FUNCTION_BLOCK FB_MER EXTENDS FB_CtrlBase IMPLEMENTS IBuffer
VAR_INPUT
	/// Sensor hanger detected
	In_bolHangerDetected: BOOL;
	/// Pin of Drive is detected
	In_bolPinDetected: BOOL;
	/// Sensors for jam detection
	In_a_bolJamSensor: ARRAY[1..cMAX_JAM_SENSORS] OF BOOL;
END_VAR
VAR
	/// Specific interface struct for public access
	SIf: T_Ctrl_SIf_MER;
	/// List of pointers to Childs
	a_pLineChildCtrl: ARRAY[0..Base_Const.cMaxNrOfChilds] OF POINTER TO FB_SLB;
	/// List of childs common interface
	a_pLineChildCIF: ARRAY[0..Base_Const.cMaxNrOfChilds] OF POINTER TO T_Ctrl_CIf;
	/// List of childs specific interface for additional parameters or cur
	a_pLineChildSIF: ARRAY[0..Base_Const.cMaxNrOfChilds] OF POINTER TO T_Ctrl_SIf_SLB;
	/// Function specific variables
	usiNumOfLines: USINT;
	usiNumOfValidPointerToLine: USINT;
	bolHangerExist: BOOL;
	bolGoToRun: BOOL;
	dinPassedTotalLineXOld: DINT;
	/// Used for counting passed hangers if "E_Typ_MER_MODE.MergeOverSetpoint" is selected.
	dinNumOfPassedHangers: DINT;
	/// Used for time measurement if "E_Typ_MER_MODE.MergeOverTime" is selected.
	udiMergingTime: UDINT;
	usiLineNumToReleaseAll: USINT;
	usiIndexToRelease: USINT;
	/// Last new position value from parent
	dinTransportPositionOld_um: DINT;
	/// Driven Way in the task
	dinDrivenWay_um: DINT;
	/// Position correction in faster Task cycletime
	dinPositionCorrection_um: DINT;
	/// Position of the section
	dinPositionSection_um: DINT;
	/// Section buffer
	a_stSectionBuffer: ARRAY[0..cusiSectionBuffer_SIZE] OF T_MER_Buffer_Sections;
	/// Edge detection of the inputs
	bolRE_HangerDetected: BOOL;
	/// Pin of Drive is detected
	bolRE_PinDetected: BOOL;
	bolModeMergeIntoTrpUsed: BOOL;
	bolSectionFree: BOOL;
	bolReleaseHanger: BOOL;
	/// Used to detect if a section is driven out
	dinPositionOfLastLine_um: DINT;
	/// Shadow copy of In_a_bolJamSensor[]
	a_bolJamSensorOnce: ARRAY[1..cMAX_JAM_SENSORS] OF BOOL;
	/// Start time of jam sensor is true
	a_udiTimeJamDetection: ARRAY[1..cMAX_JAM_SENSORS] OF UDINT;
	/// Jam at merger output detected 
	bolJamDetected: BOOL;
	/// Loop variable
	intI: INT;
	/// Simulated section length
	dinSimSectionLength_um: DINT := 510000;
	/// Simulated way to trigger section start/end
	dinSimWayTrigSection_um: DINT;
END_VAR
VAR CONSTANT
	/// sub States
	cSTA_SUB_INITIALIZED: INT := 500;
	cSTA_SUB_WAIT_FOR_CMD: INT := 502;
	cSTA_SUB_CHECK_HANGER_EXIST: INT := 504;
	cSTA_SUB_SEND_RELEASE: INT := 506;
	cSTA_SUB_SEND_RELEASE_ALL: INT := 508;
	cSTA_SUB_SEND_STOP: INT := 510;
	cSTA_SUB_WAIT_JOB_DONE: INT := 512;
	cSTA_SUB_CHECK_MERGE_CON: INT := 514;
	cSTA_SUB_WAIT_LINE_FREE: INT := 516;
	cSTA_SUB_END: INT := 518;
END_VAR

(*__________________________________________________________________________________________________
¦	
¦	Vistaprint Schweiz GmbH
¦	CH - 8401 Winterthur
¦
¦	www.vistaprint.ch - info@vistaprint.ch
¦___________________________________________________________________________________________________

Function desription:
The controller automatically merge hangers from different lines dependent time or distribution of the number of hangers.
Lines are always from controller type slide buffer FB_SLB.

History:
Version		Date			Author		Comment
---------------------------------------------------------------------------------------------------
0.00.1		05.09.2013		AVME/DSC	Start history. 
0.00.2		09.09.2013		AVME/DSC 	Integration of all merger basic functionalities. Test on simulator.
										Controller can work in 2 different main modes:
										-> "automatic", controller automatically merge hangers from different lines dependent E_Typ_MER_AUTO_MODE
										-> "on command", in case if merger work as charge controller. Release line X dependent from parent command.
0.00.3		19.09.2013		AVME/PRE	Implement new Base Concept
0.00.4		01.10.2013		AVME/DSC	Sub state machine general handling deleted. Not used anymore. Handled in Base Class.										
0.00.5		03.10.2013		AVME/PRE	Integrate new function insert Belt		
0.00.6		03.10.2013		AVME/PRE	Insert new sub state LOCK_SECTION.	
0.00.7		15.10.2013		AVME/DSC	Complete redesign of the merger "MergeIntoTrp" mode.
0.00.8		30.10.2013		AVME/DSC	Modifications for "MergeIntoTrp" mode during test at the tool. Good merging possible with drive speed = 0. (slow speed)
										Merging with higher speed not possible!				
0.00.9		08.11.2013		AVME/MRU	Stop merger if outfeed sensor detect a jam (Bugzilla Nr. 8)
0.00.10		03.12.2013		AVME/MRU	Add MaxCapacity / NumOfHangers properties
0.00.11		09.12.2013		AVME/DSC	Modification in method "checkStateAllLines".
										Special condition: In case if the child is in state ERROR and STOP is requested. Set child as checked.
										Parent controller need state STOP that automatic stop sequence can work for all other childs.
0.00.12		13.01.2014		AVME/MRU	Bugzilla ID 03: BufferFull for LineControl added

__________________________________________________________________________________________________*)


IF ((me.bolActivate) AND (THIS^.checkChildValid())) THEN // cyclic call enabled
	IF (CIf.Info.bolInitDone=FALSE) THEN // first cycle -> init
		CtrlInit();
		CIf.Info.bolInitDone := TRUE;
	ELSE
		CycleStartDuty();
	
		Always();
		
		StateMachine();
		
		CycleEndDuty();
	END_IF
END_IF;

METHOD PROTECTED sta_OFF : BOOL
// state implemetation
//--------------------------------------------------------------------------------------
// Entry action
	IF (me.StateMachine.intState<>me.StateMachine.intStateLastCycle) THEN
		me.StateMachine.intStateLastCycle := me.StateMachine.intState;
		;		
	END_IF

//--------------------------------------------------------------------------------------
// Cyclic action
	IF (me.StateMachine.intState=me.StateMachine.intStateLastCycle) THEN
		
		// Reset total counter
		SIf.Cur.dinNumOfMergedHangersTotal:= 0;
		
		// State Change Condition
		IF (me.Alarm.eActivAlmClass<>E_AlmClass.EOFF) AND (me.Alarm.eActivAlmClass<>E_AlmClass.OFF) THEN
			IF (me.intCmd=cCMD_STOP) THEN
				me.StateMachine.intStateNext := cSTA_STOPBusy;
			ELSIF (me.intCmd=cCMD_RUN) THEN 
				me.StateMachine.intStateNext := cSTA_RUNBusy;
			END_IF
		END_IF
	END_IF

//--------------------------------------------------------------------------------------
// Exit action
	IF (me.StateMachine.intState<>me.StateMachine.intStateNext) THEN
		;
	END_IF
END_METHOD

METHOD PROTECTED StateMachine : BOOL
SUPER^.StateMachine();

// main statemachine of base controller
CASE me.StateMachine.intState OF
    cSTA_STOPBusy: 
        THIS^.sta_STOPBusy();
    cSTA_STOP: 
        THIS^.sta_STOP();
	cSTA_RUNBusy: 
        THIS^.sta_RUNBusy();
    cSTA_RUN: 
        THIS^.sta_RUN();				
END_CASE;
END_METHOD

METHOD PROTECTED checkStateAllLines : BOOL
VAR_INPUT
	cSTA: INT;
END_VAR
VAR
	ii: INT;
	usiNumOfCheckedChilds: USINT;
END_VAR
// Method check input state of all lines

//Init
checkStateAllLines:= FALSE;
usiNumOfCheckedChilds:= 0;

// Loop over all childs
FOR ii:=0 TO usiNumOfLines-1 BY 1 DO
	// Check state	
	// Special condition: In case if the child is in state ERROR and STOP is requested. Set child as checked.
	// Parent controller need state STOP that automatic stop sequence can work for all other childs.
	IF (a_pLineChildCIF[ii]^.Job.intState = cSTA) OR ((a_pLineChildCIF[ii]^.Job.intState = cSTA_ERROR) AND (cSTA = cSTA_STOP)) THEN
		usiNumOfCheckedChilds:= usiNumOfCheckedChilds+1;
		SIf.Cur.a_bolChildReady[ii] := TRUE;
	ELSE
		SIf.Cur.a_bolChildReady[ii] := FALSE;		
	END_IF

END_FOR

// All states equal the input state
IF (usiNumOfCheckedChilds = usiNumOfLines) THEN
	checkStateAllLines:= TRUE;
END_IF
END_METHOD

METHOD PROTECTED getCmdState : STRING
VAR_INPUT
	intCmdState: INT;
	bolState: BOOL;
END_VAR
getCmdState := SUPER^.getCmdState(intCmdState:=intCmdState,bolState:=bolState); // get global/base defined cmds/states
IF (getCmdState='') THEN // global not defined get local
	// get string cmd/state string information in runtime
	IF (bolState=FALSE) THEN
		// cmd's
		CASE intCmdState OF
		END_CASE;
	ELSE
	
	// states
		CASE intCmdState OF	
			// SUB States
			cSTA_SUB_INITIALIZED:
				getCmdState := 'cSTA_SUB_INITIALIZED';			
			cSTA_SUB_WAIT_FOR_CMD:
				getCmdState := 'cSTA_SUB_WAIT_FOR_CMD';					
			cSTA_SUB_CHECK_HANGER_EXIST:
				getCmdState := 'cSTA_SUB_CHECK_HANGER_EXIST';
			cSTA_SUB_SEND_RELEASE:
				getCmdState := 'cSTA_SUB_SEND_RELEASE';
			cSTA_SUB_SEND_RELEASE_ALL:
				getCmdState := 'cSTA_SUB_SEND_RELEASE_ALL';	
			cSTA_SUB_SEND_STOP:
				getCmdState := 'cSTA_SUB_SEND_STOP';		
			cSTA_SUB_WAIT_JOB_DONE:
				getCmdState := 'cSTA_SUB_WAIT_JOB_DONE';
			cSTA_SUB_CHECK_MERGE_CON:
				getCmdState := 'cSTA_SUB_CHECK_MERGE_CON';
			cSTA_SUB_WAIT_LINE_FREE:
				getCmdState := 'cSTA_SUB_WAIT_LINE_FREE';	
			cSTA_SUB_END:
				getCmdState := 'cSTA_SUB_END';	
		END_CASE;
	END_IF
END_IF
END_METHOD

METHOD FB_init : BOOL
VAR_INPUT
	///if TRUE, the retain variables are initialized (warm start / cold start)
	bInitRetains: BOOL;
	///if TRUE, the instance afterwards gets moved into the copy code (online change)
	bInCopyCode: BOOL;
END_VAR
VAR
	ii: UINT;
END_VAR
//------------------------------------------------------------------------------------------------------------------------
// to manually change in new FUB implementation!!!
// define valid commands for this controller
FOR ii:= 0 TO (SIZEOF(CIf.Job.aCmdList)/SIZEOF(CIf.Job.aCmdList[0])-1) BY 1 DO
	IF (CIf.Job.aCmdList[ii].intCmd=cCMD_INITIALIZED) THEN
		// found first empty array element
		EXIT;
	END_IF
END_FOR

CIf.Job.aCmdList[ii].intCmd := cCMD_STOP;
CIf.Job.aCmdList[ii].strName := 'Stop'; 
CIf.Job.aCmdList[ii].bolAvailable := TRUE;
ii := ii +1;
CIf.Job.aCmdList[ii].intCmd := cCMD_RUN;
CIf.Job.aCmdList[ii].strName := 'Run';
CIf.Job.aCmdList[ii].bolAvailable := TRUE;

// set name of class/typ
CIf.Info.strType := 'FB_MER'; 

// set alarm class
SIf.Alm[1].eAlmClass := E_AlmClass.STOP;
SIf.Alm[1].strText := 'Invalid child pointer';
SIf.Alm[2].eAlmClass := E_AlmClass.INFO;
SIf.Alm[2].strText := 'Invalid line number. Line not exist';
SIf.Alm[3].eAlmClass := E_AlmClass.INFO;
SIf.Alm[3].strText := 'Merger waits for jam sensor free'; 


//*******************************************************************************
// initial values
//*******************************************************************************

// software configuration
CIf.SwCfg.bolExist := TRUE;
CIf.SwCfg.bolSimulation := FALSE;

// configuration
SIf.Cfg.usiMergeMainMode:= E_Typ_MER_MODE.Automatic;
SIf.Cfg.usiCountJamSensors:= 0;

// parameter
SIf.Par.udi_jamTimeout_ms:= 500;
// Default parameter for the lines are set in method InitLines
END_METHOD

METHOD PROTECTED Always : BOOL
VAR
	/// Looping variable
	intSec: INT;
END_VAR
IF (me.bolChangeBackToAUTO=TRUE) THEN // switch mode to automatic switch off controller
	//me.StateMachine.intStateNext := cSTA_OFFBusy;
	//me.bolChangeBackToAUTO := FALSE; // for cylinder no change to off when switch to automatic!!
END_IF

SUPER^.Always();

// ----------------------------------------------------------------------------------
// cyclic actions outside of statemachine
IF (me.StateMachine.intState<>cSTA_SINGLE_ANSWER) THEN
	
	//-------------------------------------------------
	// Provide current values for the parent
	//-------------------------------------------------	
	
	// Number of lines to merge, depends on how many times the method "AddLine" was called at init
	SIf.Cur.usiNumOfLinesToMerge:= usiNumOfLines;
	// Actual Item Count of this controller -> based on all lines
	SIf.Cur.dinCurrentItemCount:= THIS^.CalcSumOfItems();
	// Max. buffer capacity -> based on all lines
	SIf.Cur.dinMaxCapacity:= THIS^.CalcMaxCapacity();	
	
	
	// Check if mode "MergeIntoTrp" is configured. 
	// If one line is configured with this mode, all other lines will be set to the same mode automatically in CtrlInit. Mixed mode not possible.
	IF ((SIf.Cfg.usiMergeMainMode = E_Typ_MER_MODE.Automatic) AND (SIf.Par.a_LinePar[0].usiMergeMode = E_Typ_MER_AUTO_MODE.MergeIntoTrp)) THEN
	
		//----------------------------------------------------------------------
		// Calculate position for transport 
		//----------------------------------------------------------------------
			
		// If this task is used in a faster cycle as the parent, the driven way will be indirectly calculated (synchronized) over the transport speed.
		// If transport position changed from the parent (new value), synchronize the driven way 
		
		IF (dinTransportPositionOld_um <> SIf.Cur.dinTransportPosition_um) THEN
			dinDrivenWay_um := SIf.Cur.dinTransportPosition_um - SIf.Cur.dinTransportPositionCalc_um;
			SIf.Cur.dinTransportPositionCalc_um := SIf.Cur.dinTransportPosition_um;
			dinTransportPositionOld_um := SIf.Cur.dinTransportPosition_um;
			dinPositionCorrection_um := 0;
		ELSE
			// During the time, if there is no position change from the parent, calculate the driven way dependent the speed of transport.		
			// s = v * t
			dinDrivenWay_um := LREAL_TO_DINT(DINT_TO_LREAL(SIf.Cur.dinTransportspeed_um_s) * UDINT_TO_LREAL(me.FUBInfo.udiSample_ms) / 1000.0 );
			dinPositionCorrection_um := dinPositionCorrection_um + dinDrivenWay_um;
			SIf.Cur.dinTransportPositionCalc_um := dinTransportPositionOld_um + dinPositionCorrection_um;
		END_IF
	
	END_IF
	
END_IF

// ----------------------------------------------------------------------------------
// Always change actions in Base Library
// ----------------------------------------------------------------------------------
// overrule error always from base -> no EOFF State!! in EOFF go to OFF
IF (me.StateMachine.intStateNext = cSTA_EOFFBusy) THEN
	IF (me.StateMachine.intState=cSTA_OFF) THEN
		me.StateMachine.intStateNext := cSTA_OFF;
	ELSE // stay in OFF
		me.StateMachine.intStateNext := cSTA_OFFBusy;
	END_IF
END_IF

// Conditions Always
IF (((me.Alarm.eActivAlmClass=E_AlmClass.EOFF) OR (me.Alarm.eActivAlmClass=E_AlmClass.OFF) OR (me.intCmd=cCMD_OFF))
		 AND (me.StateMachine.intState<>cSTA_ERROR) AND (me.StateMachine.intState<>cSTA_ERRORQuit) AND
		(me.StateMachine.intState<>cSTA_OFF) AND (me.StateMachine.intState<>cSTA_OFFBusy)) THEN
	// alarm evt EOFF, OFF or cmd off
	me.StateMachine.intStateNext := cSTA_OFFBusy;
END_IF
END_METHOD

METHOD PROTECTED IoInBridge : BOOL
// digitale and analoge inputs read from hardware or forcing
SIf.In.bolHangerDetected.map := THIS^.In_bolHangerDetected;
SIf.In.bolPinDetected.map := THIS^.In_bolPinDetected;

// Read sensors for waiting if a jam is detected
FOR intI := 1 TO SIf.Cfg.usiCountJamSensors DO
	SIf.In.a_bolJamSensor[intI].map := THIS^.In_a_bolJamSensor[intI];
	IF (CIf.SwCfg.bolSimulation = FALSE) THEN
		getInBol(CIf.Job.bolIoForce,ADR(SIf.In.a_bolJamSensor[intI]));
	END_IF
END_FOR

IF (CIf.SwCfg.bolSimulation = FALSE) THEN
	getInBol(CIf.Job.bolIoForce,ADR(SIf.In.bolHangerDetected));
	getInBol(CIf.Job.bolIoForce,ADR(SIf.In.bolPinDetected));
	//ctrl.In.bol_PosSwitchBasicDefTyp.intern := getInBol(ctrl.ifc.Job.bol_Force ,ADR(ctrl.In.bol_PosSwitchBasicDefTyp);
ELSE
	//simulation of global IO
END_IF
END_METHOD

METHOD PROTECTED sta_STOPBusy : BOOL
// state implemetation
//--------------------------------------------------------------------------------------
// Entry action
	IF (me.StateMachine.intState<>me.StateMachine.intStateLastCycle) THEN
		me.StateMachine.intStateLastCycle := me.StateMachine.intState;
		
		// send command STOP to all existing line child controller.
		THIS^.CmdToAllLines(cCMD_STOP);

	END_IF

//--------------------------------------------------------------------------------------
// Cyclic action
	IF (me.StateMachine.intState=me.StateMachine.intStateLastCycle) THEN
			
		// State Change Condition
		// Check if all STOPPED
		IF (THIS^.checkStateAllLines(cSTA_STOP)) THEN
			me.StateMachine.intStateNext := cSTA_STOP;
		END_IF
	END_IF

//--------------------------------------------------------------------------------------
// Exit action
	IF (me.StateMachine.intState<>me.StateMachine.intStateNext) THEN
		;
	END_IF
END_METHOD

METHOD PROTECTED CtrlInit : BOOL
VAR
	ii: INT;
END_VAR
SUPER^.CtrlInit();

//----------------------------------------------------------------------
// Initialize all lines
//----------------------------------------------------------------------

// Method initialize all line child controller.
FOR ii:=0 TO usiNumOfLines-1 BY 1 DO	
	a_pLineChildCIF[ii] := THIS^.AddChild(a_pLineChildCtrl[ii]^);
	a_pLineChildSIF[ii] := a_pLineChildCtrl[ii]^.getCtrlSIf();
END_FOR

//----------------------------------------------------------------------
// Check about invalid configuration
//----------------------------------------------------------------------

// Check about invalid configuration of "MergeIntoTrp" mode. If one line is configured with this mode, set all other lines to the same mode.
bolModeMergeIntoTrpUsed:= FALSE;
// Check if any line is configured with "MergeIntoTrp" mode.
FOR ii:= 0 TO (usiNumOfLines-1) DO
	IF (SIf.Par.a_LinePar[ii].usiMergeMode = E_Typ_MER_AUTO_MODE.MergeIntoTrp) THEN
		// Mode is used
		bolModeMergeIntoTrpUsed:= TRUE;
		EXIT;
	END_IF
END_FOR
// Set  all other lines to "MergeIntoTrp" mode.
IF (bolModeMergeIntoTrpUsed = TRUE) THEN
	FOR ii:= 0 TO (usiNumOfLines-1) DO
		SIf.Par.a_LinePar[ii].usiMergeMode:= E_Typ_MER_AUTO_MODE.MergeIntoTrp;
	END_FOR	
END_IF

//----------------------------------------------------------------------
// Determine position of the last line
//----------------------------------------------------------------------
dinPositionOfLastLine_um:= SIf.Par.a_LinePar[usiNumOfLines-1].dinLinePosition_um;
END_METHOD

METHOD PROTECTED sta_STOP : BOOL
// state implemetation
//--------------------------------------------------------------------------------------
// Entry action
	IF (me.StateMachine.intState<>me.StateMachine.intStateLastCycle) THEN
		me.StateMachine.intStateLastCycle := me.StateMachine.intState;
		;
	END_IF

//--------------------------------------------------------------------------------------
// Cyclic action
	IF (me.StateMachine.intState=me.StateMachine.intStateLastCycle) THEN

		// State Change Condition	
		IF (me.intCmd = cCMD_RUN) THEN 
			me.StateMachine.intStateNext := cSTA_RUNBusy;
		END_IF
	END_IF

//-------------------------------------------------------------------------------------
// Exit action
	IF (me.StateMachine.intState<>me.StateMachine.intStateNext) THEN
		;
	END_IF
END_METHOD

METHOD PROTECTED IoOutBridge : BOOL
// digitale and analoge inputs read from hardware or forcing

// ... no physical outputs

IF (CIf.SwCfg.bolSimulation = FALSE) THEN
	// check interlocks to prevent damages
	IF (CIf.Job.bolIlkOverwrite=FALSE) THEN
		;
	END_IF
END_IF
END_METHOD

METHOD PROTECTED CmdToAllLines
VAR_INPUT
	cCMD: INT;
END_VAR
VAR
	ii: INT;
END_VAR
// Method send input command to all existing line child controller.
FOR ii:=0 TO usiNumOfLines-1 BY 1 DO	
	a_pLineChildCIF[ii]^.Job.intACmd:= cCMD;
END_FOR
END_METHOD

METHOD PROTECTED sta_RUN : BOOL
VAR
	/// Looping variable
	intSec: INT;
END_VAR
// state implemetation
//--------------------------------------------------------------------------------------
// Entry action
	IF (me.StateMachine.intState<>me.StateMachine.intStateLastCycle) THEN
		me.StateMachine.intStateLastCycle := me.StateMachine.intState;	
		;	
	END_IF

//--------------------------------------------------------------------------------------
// Cyclic action
	IF (me.StateMachine.intState=me.StateMachine.intStateLastCycle) THEN
			
		//-------------------------------------------------
		// Handling to merge into a transport belt
		//-------------------------------------------------	
		
		// Check if mode "MergeIntoTrp" is configured. 
		// If one line is configured with this mode, all other lines will be set to the same mode automatically in CtrlInit. Mixed mode not possible.
		IF ((SIf.Cfg.usiMergeMainMode = E_Typ_MER_MODE.Automatic) AND (SIf.Par.a_LinePar[0].usiMergeMode = E_Typ_MER_AUTO_MODE.MergeIntoTrp)) THEN
						
			//----------------------------------------------------------------------
			// Set the section start and end positions (triggered by pin sensor)
			//----------------------------------------------------------------------
			
			// Simulation of section start and end
			IF (CIf.SwCfg.bolSimulation = TRUE) THEN		
				SIf.In.bolPinDetected.intern:= FALSE;
				
				IF (dinSimWayTrigSection_um >= dinSimSectionLength_um) THEN
					dinSimWayTrigSection_um:= 0;
					// Set true for one cycle
					SIf.In.bolPinDetected.intern:= TRUE;
				END_IF
				// Increase position		
				dinSimWayTrigSection_um:= dinSimWayTrigSection_um + dinDrivenWay_um;
			END_IF
					
			// Wait for positive edge of the pin sensor (pin detected)
			IF (SIf.In.bolPinDetected.intern = TRUE) AND (bolRE_PinDetected = FALSE) THEN
				bolRE_PinDetected := TRUE;
					
				// Loop over section buffer
				FOR intSec := 0 TO cusiSectionBuffer_SIZE DO
					
					// If start position already set
					IF (a_stSectionBuffer[intSec].usiState = 1) THEN						
						// Set end position of the section
						a_stSectionBuffer[intSec].dinSecEndPos:= 0 - SIf.Par.dinPinLenght_um;
						a_stSectionBuffer[intSec].usiState:= 2;
					END_IF
					
					// Free buffer element  
					IF (a_stSectionBuffer[intSec].usiState = 0) THEN			
						// Set start position of the section
						a_stSectionBuffer[intSec].dinSecStartPos:= 0 - SIf.Par.dinPinLenght_um;
						a_stSectionBuffer[intSec].usiState:= 1;
						EXIT;									  
					END_IF
													
				END_FOR
					
			ELSIF (SIf.In.bolPinDetected.intern = FALSE) AND (bolRE_PinDetected = TRUE) THEN
				bolRE_PinDetected := FALSE;
			END_IF
			
			//----------------------------------------------------------------------
			// Set section engaged (hanger in section)
			//----------------------------------------------------------------------
			
			// Wait for positive edge of the hanger sensor
			IF (SIf.In.bolHangerDetected.intern = TRUE) AND (bolRE_HangerDetected = FALSE) THEN
				bolRE_HangerDetected := TRUE;
					
				// Loop over section buffer to mark buffer element with 3 = section engaged (hanger in section detected by hanger sensor)
				FOR intSec := 0 TO cusiSectionBuffer_SIZE-1 DO		
					
					// Prio 1: Normal sequence.
					IF (SIf.Par.dinHangerSensorPosition_um < a_stSectionBuffer[intSec].dinSecStartPos) AND  
						(SIf.Par.dinHangerSensorPosition_um > (a_stSectionBuffer[intSec].dinSecEndPos - SIf.Par.dinPinLenght_um)) THEN	
							// Mark the buffer element with 3 = section engaged (hanger in section detected by hanger sensor)
							a_stSectionBuffer[intSec].usiState:= 3;
						EXIT;
					
					// Prio 2: If range is not accurately recognized mark buffer element X and X +1.
					ELSIF (SIf.Par.dinHangerSensorPosition_um < a_stSectionBuffer[intSec].dinSecEndPos) AND  
						(SIf.Par.dinHangerSensorPosition_um > a_stSectionBuffer[intSec+1].dinSecStartPos) THEN	
							// Mark the buffer element with 3 = section engaged (hanger in section detected by hanger sensor)
							a_stSectionBuffer[intSec].usiState:= 3;
							a_stSectionBuffer[intSec+1].usiState:= 3;
						EXIT;
					END_IF		
						
				END_FOR	
					
			ELSIF (SIf.In.bolHangerDetected.intern = FALSE) AND (bolRE_HangerDetected = TRUE) THEN
				bolRE_HangerDetected := FALSE;
			END_IF	
				
			//----------------------------------------------------------------------
			// Buffer tracking 
			//----------------------------------------------------------------------
			
			// Move all buffer elements 1 down if hanger was released. State will be set to "0" in state RUN if a hanger is released.
			// Also check if a section is driven out!			
			IF (a_stSectionBuffer[0].usiState = 0) OR (a_stSectionBuffer[0].dinSecEndPos > (dinPositionOfLastLine_um + SIf.Par.dinSectionLenght_um))THEN
				// Loop every buffer element 1 Down
				FOR intSec := 0 TO cusiSectionBuffer_SIZE-1 DO			
					a_stSectionBuffer[intSec].dinSecStartPos := a_stSectionBuffer[intSec+1].dinSecStartPos;
					a_stSectionBuffer[intSec].dinSecEndPos := a_stSectionBuffer[intSec+1].dinSecEndPos;
					a_stSectionBuffer[intSec].dinTrigStartPos := a_stSectionBuffer[intSec+1].dinTrigStartPos;
					a_stSectionBuffer[intSec].dinTrigEndPos := a_stSectionBuffer[intSec+1].dinTrigEndPos;
					a_stSectionBuffer[intSec].usiState := a_stSectionBuffer[intSec+1].usiState;
				END_FOR		
				a_stSectionBuffer[intSec].dinSecStartPos := 0;
				a_stSectionBuffer[intSec].dinSecEndPos := 0;
				a_stSectionBuffer[intSec].dinTrigStartPos := 0;
				a_stSectionBuffer[intSec].dinTrigEndPos := 0;
				a_stSectionBuffer[intSec].usiState := 0;
			END_IF
			
			//----------------------------------------------------------------------
			// Increase positions
			//----------------------------------------------------------------------
				
			// Increase the buffer positions
			FOR intSec := 0 TO cusiSectionBuffer_SIZE DO
				
				IF (a_stSectionBuffer[intSec].usiState = 1) THEN
					// Section start/end
					a_stSectionBuffer[intSec].dinSecStartPos:= a_stSectionBuffer[intSec].dinSecStartPos + dinDrivenWay_um;
					// Trigger start/end
					a_stSectionBuffer[intSec].dinTrigStartPos:= a_stSectionBuffer[intSec].dinSecStartPos - SIf.Par.dinTrigStartOffset_um;
					a_stSectionBuffer[intSec].dinTrigEndPos:= a_stSectionBuffer[intSec].dinSecStartPos - SIf.Par.dinTrigEndOffset_um;	
					
				ELSIF (a_stSectionBuffer[intSec].usiState >= 2) THEN
					// Section start/end
					a_stSectionBuffer[intSec].dinSecStartPos:= a_stSectionBuffer[intSec].dinSecStartPos + dinDrivenWay_um;
					a_stSectionBuffer[intSec].dinSecEndPos:= a_stSectionBuffer[intSec].dinSecEndPos + dinDrivenWay_um;
					// Trigger start/end
					a_stSectionBuffer[intSec].dinTrigStartPos:= a_stSectionBuffer[intSec].dinSecStartPos - SIf.Par.dinTrigStartOffset_um;
					a_stSectionBuffer[intSec].dinTrigEndPos:= a_stSectionBuffer[intSec].dinSecStartPos - SIf.Par.dinTrigEndOffset_um;				
				END_IF
				
			END_FOR	
			
		END_IF
	
		
		// Check States for parent information
		THIS^.checkStateAllLines(cSTA_RUN);

		// Check jam detection
		bolJamDetected := FALSE;
		FOR intI := 1 TO SIf.Cfg.usiCountJamSensors DO
			// Start jam timer
			IF ((SIf.In.a_bolJamSensor[intI].intern = TRUE) AND (a_bolJamSensorOnce[intI] = FALSE)) THEN
				a_bolJamSensorOnce[intI]:= TRUE;
				a_udiTimeJamDetection[intI]:= me.StateMachine.udiTimeInState_ms;
			// Stop jam timer
			ELSIF ((SIf.In.a_bolJamSensor[intI].intern = FALSE) AND (a_bolJamSensorOnce[intI] = TRUE)) THEN
				a_bolJamSensorOnce[intI]:= FALSE;
				//a_bolJamDetected[intI] := FALSE;
			// Set flag if neccessary
			ELSIF ((SIf.In.a_bolJamSensor[intI].intern = TRUE) AND (a_bolJamSensorOnce[intI] = TRUE)) THEN
				IF (me.StateMachine.udiTimeInState_ms > a_udiTimeJamDetection[intI] + SIf.Par.udi_jamTimeout_ms) THEN
					bolJamDetected := TRUE;
				END_IF
			END_IF
		END_FOR
	
		//----------------------------------------------------------------------------------------
		// Substates for merging lines dependent time or distribution of the number of hangers
		//----------------------------------------------------------------------------------------
		CASE me.SubStateMachine.intState OF
	
			//-----------------------------------------------
			// INITIALIZE 					(MODE: All modes)
			//-----------------------------------------------
			cSTA_SUB_INITIALIZED:
			
				// Check configured main mode
				CASE SIf.Cfg.usiMergeMainMode OF	
				
					// Mode - Automatic
					E_Typ_MER_MODE.Automatic:		
						me.SubStateMachine.intStateNext := cSTA_SUB_CHECK_HANGER_EXIST;					
									
					// Mode - OnCommand	
					E_Typ_MER_MODE.OnCommand:		
						me.SubStateMachine.intStateNext := cSTA_SUB_WAIT_FOR_CMD;
														
				END_CASE
			
			//-----------------------------------------------
			// WAIT FOR COMMAND 			(MODE: OnCommand)
			//-----------------------------------------------	
			cSTA_SUB_WAIT_FOR_CMD:
			
				// Wait for command to release all
				IF (me.intCmd=SLB_CmdState.cCMD_RELEASE_ALL) THEN
					// Check about valid line number
					IF ((SIf.Par.usiLineNumToReleaseAll = 0) OR (SIf.Par.usiLineNumToReleaseAll > usiNumOfLines)) THEN
						// Invalid line	
						// SIf.Alm[2].strText := 'Invalid line number. Line not exist'; 
						pfbAlarmCtrl^.setAlarm(CIf.Info.intCtrlId,2,0,ADR(SIf.Alm),E_AlmState.RST,CIf.Job.eMe_ActivAlmClass);		
					ELSE
						// Valid line	
						usiLineNumToReleaseAll:= SIf.Par.usiLineNumToReleaseAll-1;
						me.SubStateMachine.intStateNext := cSTA_SUB_SEND_RELEASE_ALL;
					END_IF
						
				END_IF
				
			//-----------------------------------------------
			// CHECK HANGER EXIST 			(MODE: Automatic)     
			//-----------------------------------------------
			cSTA_SUB_CHECK_HANGER_EXIST:
				// Entry action
				IF (me.SubStateMachine.intState<>me.SubStateMachine.intStateLastCycle) THEN
					me.SubStateMachine.intStateLastCycle := me.SubStateMachine.intState;							
					;						
				END_IF
		
				// Init
				bolReleaseHanger:= FALSE;
				bolSectionFree := FALSE;
						
				// Check if mode "MergeIntoTrp" is configured.
				IF (SIf.Par.a_LinePar[usiIndexToRelease].usiMergeMode = E_Typ_MER_AUTO_MODE.MergeIntoTrp) THEN
					FOR intSec := 0 TO cusiSectionBuffer_SIZE DO
						// Check if the current line position is within the trigger window to release the hanger
						IF ((SIf.Par.a_LinePar[usiIndexToRelease].dinLinePosition_um < a_stSectionBuffer[intSec].dinTrigStartPos)
							AND (SIf.Par.a_LinePar[usiIndexToRelease].dinLinePosition_um > a_stSectionBuffer[intSec].dinTrigEndPos)
							AND (a_stSectionBuffer[intSec].usiState = 2)) THEN
								// Section is free, hanger can be released
								bolSectionFree := TRUE;	
								EXIT;
						END_IF
					END_FOR					
				END_IF
					
				// Check hanger exists on line
				IF (((a_pLineChildSIF[usiIndexToRelease]^.Cur.bolHangerDetected=TRUE) AND (SIf.Par.a_LinePar[usiIndexToRelease].usiMergeMode <> E_Typ_MER_AUTO_MODE.MergeIntoTrp)) OR
					((a_pLineChildSIF[usiIndexToRelease]^.Cur.bolHangerDetected=TRUE) AND (bolSectionFree = TRUE) AND (SIf.Par.a_LinePar[usiIndexToRelease].usiMergeMode = E_Typ_MER_AUTO_MODE.MergeIntoTrp))) THEN		

					IF (SIf.Par.a_LinePar[usiIndexToRelease].usiMergeMode = E_Typ_MER_AUTO_MODE.MergeIntoTrp) THEN
						// Mark the buffer element with 4 = hanger released (section engaged)
						a_stSectionBuffer[intSec].usiState:= 4;	
					END_IF
					bolReleaseHanger:= TRUE;
					
				ELSE		
					// No hanger on this line, check next
					IF (usiIndexToRelease < (usiNumOfLines-1)) THEN
						// Inc. index to next line
						usiIndexToRelease:= usiIndexToRelease + 1;	
					ELSE
						usiIndexToRelease:= 0;
					END_IF
				END_IF			

		
				// State Change Condition
				IF (bolReleaseHanger=TRUE) THEN
					me.SubStateMachine.intStateNext := cSTA_SUB_SEND_RELEASE;
					// Reset counter and timer
					dinNumOfPassedHangers:=0;
					udiMergingTime:=0;
				END_IF
						
			//-----------------------------------------------
			// SEND RELEASE					(MODE: Automatic)
			//-----------------------------------------------
			cSTA_SUB_SEND_RELEASE:		
	
				// Send release command to line X (trigger command)
				a_pLineChildCIF[usiIndexToRelease]^.Job.intACmd:= STB_CmdState.cCMD_RELEASE;				
				
				// State Change Condition
				IF(TRUE)THEN
					me.SubStateMachine.intStateNext := cSTA_SUB_WAIT_JOB_DONE;					
				END_IF	
						
			//-----------------------------------------------
			// SEND RELEASE	ALL				(MODE: OnCommand)
			//-----------------------------------------------
			cSTA_SUB_SEND_RELEASE_ALL:
			
				// Send release all command to line X
				a_pLineChildCIF[usiLineNumToReleaseAll]^.Job.intACmd:= STB_CmdState.cCMD_RELEASE_ALL;				
				
				// State Change Condition
				IF(TRUE)THEN
					me.SubStateMachine.intStateNext := cSTA_SUB_WAIT_JOB_DONE;					
				END_IF		
					
			//-----------------------------------------------
			// WAIT JOB DONE				(MODE: All modes)
			//-----------------------------------------------
			cSTA_SUB_WAIT_JOB_DONE:
		
				// Check configured main mode
				CASE SIf.Cfg.usiMergeMainMode OF	
				
					// Mode - Automatic
					E_Typ_MER_MODE.Automatic:
						// State Change Condition
						// Wait until job done
						IF(a_pLineChildCIF[usiIndexToRelease]^.Job.intACmd = cSTA_DONE)THEN									
							IF (SIf.Par.a_LinePar[usiIndexToRelease].usiMergeMode = E_Typ_MER_AUTO_MODE.MergeIntoTrp) THEN							
								me.SubStateMachine.intStateNext := cSTA_SUB_WAIT_LINE_FREE;							
							ELSE
								me.SubStateMachine.intStateNext := cSTA_SUB_CHECK_MERGE_CON;
							END_IF																					
						END_IF	
									
					// Mode - OnCommand	
					E_Typ_MER_MODE.OnCommand:
						// State Change Condition
						// Wait until release all
						IF(a_pLineChildCIF[usiLineNumToReleaseAll]^.Job.intState = SLB_CmdState.cCMD_RELEASE_ALL)THEN				
							me.SubStateMachine.intStateNext := cSTA_SUB_SEND_STOP;																
						END_IF
						
				END_CASE
							
			//-----------------------------------------------
			// SEND STOP					(MODE: OnCommand)
			//-----------------------------------------------
			cSTA_SUB_SEND_STOP:
			
				// Send stop command to line X
				a_pLineChildCIF[usiLineNumToReleaseAll]^.Job.intACmd:=cCMD_RUN;				
				
				// State Change Condition
				IF(a_pLineChildCIF[usiLineNumToReleaseAll]^.Job.intState=cSTA_RUN)THEN
					me.SubStateMachine.intStateNext := cSTA_SUB_WAIT_LINE_FREE;					
				END_IF	
								
			//-----------------------------------------------
			// CHECK MERGE CONDITIONS		(MODE: Automatic)
			//-----------------------------------------------
			cSTA_SUB_CHECK_MERGE_CON:
				// Entry action
				IF (me.SubStateMachine.intState<>me.SubStateMachine.intStateLastCycle) THEN
					me.SubStateMachine.intStateLastCycle := me.SubStateMachine.intState;							
					;						
				END_IF
					
				// Count the passed hangers from current line X
				IF (a_pLineChildSIF[usiIndexToRelease]^.Cur.dinHangersPassedTotal <> dinPassedTotalLineXOld) THEN
					// Count passed hangers if "E_Typ_MER_AUTO_MODE.MergeOverSetpoint" is selected.				
					dinNumOfPassedHangers:= dinNumOfPassedHangers + a_pLineChildSIF[usiIndexToRelease]^.Cur.uinNumOfHangersPerPulseFirstZone;			
					// Calculate merged hangers total
					SIf.Cur.dinNumOfMergedHangersTotal:= SIf.Cur.dinNumOfMergedHangersTotal + a_pLineChildSIF[usiIndexToRelease]^.Cur.uinNumOfHangersPerPulseFirstZone;									
				END_IF
				dinPassedTotalLineXOld:= a_pLineChildSIF[usiIndexToRelease]^.Cur.dinHangersPassedTotal;
		
					
				// State Change Condition
				IF (a_pLineChildSIF[usiIndexToRelease]^.Cur.bolHangerDetected=FALSE) THEN	// No hanger exist
					me.SubStateMachine.intStateNext := cSTA_SUB_WAIT_LINE_FREE;				
				ELSIF ((SIf.Par.a_LinePar[usiIndexToRelease].usiMergeMode = E_Typ_MER_AUTO_MODE.MergeOverTime) AND (udiMergingTime >= SIf.Par.a_LinePar[usiIndexToRelease].udiMergingTime_ms)) THEN
					me.SubStateMachine.intStateNext := cSTA_SUB_WAIT_LINE_FREE;				
				ELSIF ((SIf.Par.a_LinePar[usiIndexToRelease].usiMergeMode = E_Typ_MER_AUTO_MODE.MergeOverSetpoint) AND (dinNumOfPassedHangers >= SIf.Par.a_LinePar[usiIndexToRelease].uinNumOfHangersToMerge)) THEN
					me.SubStateMachine.intStateNext := cSTA_SUB_WAIT_LINE_FREE;							
				ELSIF ((SIf.Par.a_LinePar[usiIndexToRelease].usiMergeMode = E_Typ_MER_AUTO_MODE.MergeOverTime) AND (udiMergingTime < SIf.Par.a_LinePar[usiIndexToRelease].udiMergingTime_ms)) THEN
					me.SubStateMachine.intStateNext := cSTA_SUB_SEND_RELEASE;					
				ELSIF ((SIf.Par.a_LinePar[usiIndexToRelease].usiMergeMode = E_Typ_MER_AUTO_MODE.MergeOverSetpoint) AND (dinNumOfPassedHangers < SIf.Par.a_LinePar[usiIndexToRelease].uinNumOfHangersToMerge)) THEN
					me.SubStateMachine.intStateNext := cSTA_SUB_SEND_RELEASE;	
				END_IF
	
			//-----------------------------------------------
			// WAIT UNTIL LINE IS FREE		(MODE: All modes)
			//-----------------------------------------------
			cSTA_SUB_WAIT_LINE_FREE:

				IF (bolJamDetected	= TRUE) THEN // Line is not free, jam detected
					// SIf.Alm[3].strText := 'Merger waits for jam sensor free';
					pfbAlarmCtrl^.setAlarm(CIf.Info.intCtrlId,3,0,ADR(SIf.Alm),E_AlmState.RST,CIf.Job.eMe_ActivAlmClass);				
				ELSE				
					// Check configured main mode
					CASE SIf.Cfg.usiMergeMainMode OF	
					
						// Mode - Automatic
						E_Typ_MER_MODE.Automatic:
							// State Change Condition
							IF (me.SubStateMachine.udiTimeInState_ms > SIf.Par.a_LinePar[usiIndexToRelease].udiWaitTimeLineFree_ms) OR 
								(SIf.Par.a_LinePar[usiIndexToRelease].usiMergeMode = E_Typ_MER_AUTO_MODE.MergeIntoTrp) THEN
								IF(me.intCmd=cCMD_STOP)THEN
									// Go to end
									me.SubStateMachine.intStateNext := cSTA_SUB_END;
								ELSE
									// Merging cycle line X complete
									IF (usiIndexToRelease < (usiNumOfLines-1)) THEN						
										// Inc. index to next line
										usiIndexToRelease:= usiIndexToRelease + 1;	
									ELSE
										usiIndexToRelease:= 0;
									END_IF
									
									// Go on with automatic cycle
									me.SubStateMachine.intStateNext := cSTA_SUB_CHECK_HANGER_EXIST;					
								END_IF		
							END_IF
									
						// Mode - OnCommand	
						E_Typ_MER_MODE.OnCommand:
							// State Change Condition
							IF (me.SubStateMachine.udiTimeInState_ms > SIf.Par.a_LinePar[usiLineNumToReleaseAll].udiWaitTimeLineFree_ms) THEN												
								// Update merged hangers total -> After release all, use passed package 
								SIf.Cur.dinNumOfMergedHangersTotal:= SIf.Cur.dinNumOfMergedHangersTotal + a_pLineChildSIF[usiLineNumToReleaseAll]^.Cur.dinHangersPassedPackage;			
								
								IF(me.intCmd=cCMD_STOP)THEN
									// Go to end
									me.SubStateMachine.intStateNext := cSTA_SUB_END;
								ELSE
									//Set "Job done" for parent
									CIf.Job.intACmd:=cSTA_DONE;
									me.SubStateMachine.intStateNext := cSTA_SUB_WAIT_FOR_CMD;
								END_IF								
							END_IF
							
					END_CASE
				END_IF
			//-----------------------------------------------
			// END							(MODE: All modes)
			//-----------------------------------------------
			cSTA_SUB_END:
			     // ... do nothing
		
		END_CASE

		// Timer handling for merging time
		udiMergingTime:= udiMergingTime + me.FUBInfo.udiSample_ms;
			
		// State Change Condition
		IF ((me.intCmd=cCMD_STOP) AND ((me.SubStateMachine.intState=cSTA_SUB_END) OR (me.SubStateMachine.intState=cSTA_SUB_CHECK_HANGER_EXIST) OR (me.SubStateMachine.intState=cSTA_SUB_WAIT_FOR_CMD) OR (me.SubStateMachine.intState=cSTA_SUB_WAIT_LINE_FREE))) THEN
			me.StateMachine.intStateNext := cSTA_STOPBusy;
		END_IF
	END_IF

//--------------------------------------------------------------------------------------
// Exit action
	IF (me.StateMachine.intState<>me.StateMachine.intStateNext) THEN
		;
	END_IF
END_METHOD

METHOD getCtrlSIf : POINTER TO T_Ctrl_SIf_MER
getCtrlSIf := ADR(SIf);
END_METHOD

METHOD AddLine
VAR_INPUT
	p_Line: POINTER TO FB_SLB;
END_VAR

// Method add the pointer address of the line child controller to the array list.
IF (usiNumOfLines <= (Base_Const.cMaxNrOfChilds-1)) THEN
	// Add line child controller to list
	a_pLineChildCtrl[usiNumOfLines] := p_Line;
	// Inc. number of lines
	usiNumOfLines:= usiNumOfLines+1;
	// Check if the pointer is valid
	IF (p_Line<>0) THEN
		usiNumOfValidPointerToLine:= usiNumOfValidPointerToLine+1;
	END_IF
END_IF
END_METHOD

METHOD PROTECTED CalcMaxCapacity : DINT
VAR
	ii: INT;
	dinSumMaxCapacity: DINT;
END_VAR
// Method calculate the sum of max. capacities from all lines and return the result.

//Init
CalcMaxCapacity:= 0;
dinSumMaxCapacity:= 0;

// Loop over all childs
FOR ii:=0 TO usiNumOfLines-1 BY 1 DO
	// Build sum of all lines		
	dinSumMaxCapacity:= dinSumMaxCapacity + a_pLineChildSIF[ii]^.Cur.dinMaxCapacity; 	
END_FOR

// Return result
CalcMaxCapacity:= dinSumMaxCapacity;
END_METHOD

METHOD PROTECTED sta_RUNBusy : BOOL
VAR
	ii: INT;
END_VAR
// state implemetation
//--------------------------------------------------------------------------------------
// Entry action
	IF (me.StateMachine.intState<>me.StateMachine.intStateLastCycle) THEN
		me.StateMachine.intStateLastCycle := me.StateMachine.intState;
	
		bolGoToRun:= FALSE;
		usiIndexToRelease:= 0;
		
		// Initialize sub state machine
		me.SubStateMachine.intState:= cSTA_SUB_INITIALIZED; 
		me.SubStateMachine.intStateNext:= cSTA_SUB_INITIALIZED;
		
	END_IF

//--------------------------------------------------------------------------------------
// Cyclic action
	IF (me.StateMachine.intState=me.StateMachine.intStateLastCycle) THEN
			
		// Check if mode "MergeIntoTrp" is configured. 
		IF ((SIf.Cfg.usiMergeMainMode = E_Typ_MER_MODE.Automatic) AND (SIf.Par.a_LinePar[0].usiMergeMode = E_Typ_MER_AUTO_MODE.MergeIntoTrp)) THEN
			// Clear section buffer
			FOR ii := 0 TO cusiSectionBuffer_SIZE DO
				a_stSectionBuffer[ii].dinSecStartPos := 0;
				a_stSectionBuffer[ii].dinSecEndPos := 0;
				a_stSectionBuffer[ii].dinTrigStartPos := 0;
				a_stSectionBuffer[ii].dinTrigEndPos := 0;
				a_stSectionBuffer[ii].usiState := 0;				
			END_FOR
		END_IF
		
		// Check configured main mode
		CASE SIf.Cfg.usiMergeMainMode OF	
		
			// Mode - Automatic
			E_Typ_MER_MODE.Automatic:
			
				// send command RUN to all existing line child controller.
				THIS^.CmdToAllLines(cCMD_RUN);
				
				// State Change Condition
				// Check if all childs in "RUN", ready for release hanger 
				IF(THIS^.checkStateAllLines(cSTA_RUN))THEN
					bolGoToRun:= TRUE;			
				END_IF	
		
			// Mode - OnCommand	
			E_Typ_MER_MODE.OnCommand:
			
				// send command STOP to all existing line child controller.
				THIS^.CmdToAllLines(cCMD_RUN);
				
				// State Change Condition
				// Check if all childs stopped, ready for new command 
				IF(THIS^.checkStateAllLines(cSTA_RUN))THEN
					bolGoToRun:= TRUE;					
				END_IF	
			
		END_CASE

	
		// State Change Condition	
		IF (bolGoToRun=TRUE) THEN
			me.StateMachine.intStateNext := cSTA_RUN;		
		END_IF

	END_IF

//--------------------------------------------------------------------------------------
// Exit action
	IF (me.StateMachine.intState<>me.StateMachine.intStateNext) THEN
		;
	END_IF
END_METHOD

METHOD PROTECTED checkChildValid : BOOL
IF (usiNumOfLines = usiNumOfValidPointerToLine) THEN
	checkChildValid:= TRUE;
ELSE
	checkChildValid:= FALSE;
	// Invalid child pointer
	IF (usiNumOfLines <> usiNumOfValidPointerToLine) THEN
		// SIf.Alm[1].strText := 'Invalid child pointer'; 
		pfbAlarmCtrl^.setAlarm(CIf.Info.intCtrlId,1,0,ADR(SIf.Alm),E_AlmState.RST,CIf.Job.eMe_ActivAlmClass);	
	END_IF
END_IF
END_METHOD

METHOD PROTECTED CalcSumOfItems : DINT
VAR
	ii: INT;
	dinSumOfItems: DINT;
END_VAR
// Method calculate the sum of hangers from all lines and return the result.

//Init
CalcSumOfItems:= 0;
dinSumOfItems:= 0;

// Loop over all childs
FOR ii:=0 TO usiNumOfLines-1 BY 1 DO
	// Build sum of all zones		
	dinSumOfItems:= dinSumOfItems + a_pLineChildSIF[ii]^.Cur.dinNumOfHangersInBuffer; 	
END_FOR

// Return result
CalcSumOfItems:= dinSumOfItems;
END_METHOD

METHOD checkChildAlmClass : BOOL
//------------------------------------------------------------------------------------------------------
// check child alarm classes
// set me alarm class active if at least one child has an EOFF
IF CheckAllChildAlmClass(E_AlmClass.EOFF) THEN
	CIf.Job.eMe_ActivAlmClass := E_AlmClass.EOFF;
	me.Alarm.bolfp := TRUE;
ELSIF CheckAllChildAlmClass(E_AlmClass.OFF) THEN
	CIf.Job.eMe_ActivAlmClass := E_AlmClass.OFF;
	me.Alarm.bolfp := TRUE;
ELSIF CheckAllChildAlmClass(E_AlmClass.STOP) THEN  // FB_MER needs alarm class STOP
	CIf.Job.eMe_ActivAlmClass := E_AlmClass.STOP;
	me.Alarm.bolfp := TRUE;
ELSE
	IF (me.Alarm.bolfp) THEN
		CIf.Job.eMe_ActivAlmClass := E_AlmClass.NONE; // no reset necessary
		me.Alarm.bolfp := FALSE;
	END_IF
END_IF

//------------------------------------------------------------------------------------------------------
// set alarm class parent of childs
//------------------------------------------------------------------------------------------------------
// set alarm class parent of childs in the case of a parent EOFF or me=OFF or EOFF
IF (CIf.Job.eParent_ActivAlmClass=E_AlmClass.EOFF) THEN
	SetAllChildAlmClass(CIf.Job.eParent_ActivAlmClass);
ELSIF(CIf.Job.eMe_ActivAlmClass=E_AlmClass.EOFF) OR (CIf.Job.eMe_ActivAlmClass=E_AlmClass.OFF) THEN
	SetAllChildAlmClass(CIf.Job.eMe_ActivAlmClass);
ELSE
	// no important alarm for child active
	SetAllChildAlmClass(E_AlmClass.NONE);
END_IF
END_METHOD

PROPERTY NumOfHangers : DINT
GET
NumOfHangers:= SIf.Cur.dinCurrentItemCount;
END_GET
END_PROPERTY

PROPERTY MaxCapacity : DINT
GET
MaxCapacity:= SIf.Cur.dinMaxCapacity;
END_GET
END_PROPERTY

PROPERTY BufferFull : BOOL
GET
BufferFull:= False;
END_GET
END_PROPERTY

END_FUNCTION_BLOCK

(* stored: Version 1.1.0.1, ProductVersion 3.1.0.19
   POU FB_MER: Id {81e1f74f-aae1-42cf-9873-cf8a29e6c322}
   Method sta_OFF: Id {a2d4d6b4-8e17-4352-8516-af7ed8f02a80}
   Method StateMachine: Id {7ba70d8e-77b0-4e5d-9e00-77a064cba4f8}
   Method checkStateAllLines: Id {982b8bae-f8ff-4f28-930f-49ca1cdf1f51}
   Method getCmdState: Id {9b91bf69-7311-405c-8aa0-b2ed0cc6f6af}
   Method FB_init: Id {c4d218ea-a65b-4e13-aa14-4b29912961d5}
   Method Always: Id {1da635e9-7b39-44bb-8869-10a4027ca53f}
   Method IoInBridge: Id {0d0a73b2-64e0-4a3e-98e4-3985a499f182}
   Method sta_STOPBusy: Id {e73347e6-d359-4d6e-9cf3-09d28c932c40}
   Method CtrlInit: Id {483de46a-1813-4732-ba54-429bc4b8410d}
   Method sta_STOP: Id {7713e70e-ad89-49ba-aa03-fe8e0b98321d}
   Method IoOutBridge: Id {2c78accc-afc7-4d90-acf7-275a5a13ccc1}
   Method CmdToAllLines: Id {3b97476f-9fb7-4f1d-9b47-9554ee126bdf}
   Method sta_RUN: Id {9fda181c-f474-4ad2-b574-65ed50a3091e}
   Method getCtrlSIf: Id {792d7e83-d67a-435f-9cef-02393e414a15}
   Method AddLine: Id {d272e310-154a-4706-917e-47bd91856013}
   Method CalcMaxCapacity: Id {7cc9409e-d41f-4a8b-b36d-ebdd2f7429d5}
   Method sta_RUNBusy: Id {5b4a2819-60e3-4465-bb6e-50cef987fe85}
   Method checkChildValid: Id {1ad30143-7a77-4e83-8f6f-af25c5ef12f7}
   Method CalcSumOfItems: Id {115a0ded-0390-40d0-8cf8-cd15a5839728}
   Method checkChildAlmClass: Id {76218c07-bdad-4421-b652-7a3736fca00c}
   Property NumOfHangers: Id {070aa852-d01d-4086-a7f9-d5ac0fe3831f}
   Get Get: Id {df6222c4-8f3d-42a0-8c26-c94ff8399322}
   Property MaxCapacity: Id {7a147946-14e1-4a40-a5f2-cb6f59ea8dfb}
   Get Get: Id {74eb6a77-8cdd-41ba-9c15-abcf705e6619}
   Property BufferFull: Id {201eac71-4233-43f6-b777-56ce7f3e21a0}
   Get Get: Id {a48a61b8-1194-4725-9144-9816681c195b} *)
